FUNCTION_BLOCK Test_TimeAsString_IncludesLeadingZeros EXTENDS TUnitTestBase
VAR
END_VAR

METHOD  Execute
VAR_INST
    TimeStruct : TIMESTRUCT := (wHour := 6, wMinute := 5, wSecond := 4);
END_VAR
Assertion.AssertEquals_STRING(
    Expected := '06:05:04',
    Actual   := F_TimeAsString(TimeStruct),
    ObjectName := _TestName,
    VariableName  := 'F_TimeAsString(TimeStruct)');


Test_Finished();
END_METHOD

END_FUNCTION_BLOCK

(* stored: Version 1.1.0.1, ProductVersion 3.1.4024.3
   POU Test_TimeAsString_IncludesLeadingZeros: Id {a848e1a0-6f7e-4283-a08e-78011e686f1e}, SpecialFunc None
   Method Execute: Id {2434403a-5dc7-48fc-9b97-4d9a9c6685e7} *)
